# B&R Automation Studio project brse_dtf
Automation Studio 6.5.0.306; technology packages: OpcUaCs 6.5.0

## Configuration ARM

CPU X20CP0484, AutomationRuntime 6.5.1, Build 11.3.0, Vc 6.0.0

### Hardware
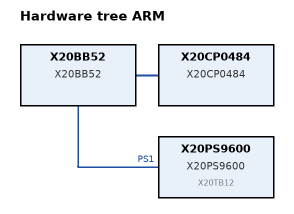
```
X20BB52 : X20BB52 v1.2.0.0
X20CP0484 : X20CP0484 v1.8.1.0  [SL -> X20BB52.SL1]
  TimerDeviceType = SWIOTIMER
  Cyclic1Duration = 10000
  Cyclic1Tolerance = 10000
  Cyclic2Duration = 20000
  Cyclic2Tolerance = 20000
  Cyclic3Duration = 50000
  Cyclic3Tolerance = 50000
  Cyclic4Duration = 100000
  Cyclic4Tolerance = 100000
  Cyclic5Duration = 200000
  Cyclic5Tolerance = 200000
  Cyclic6Duration = 500000
  Cyclic6Tolerance = 500000
  Cyclic7Duration = 1000000
  Cyclic7Tolerance = 1000000
  Cyclic8Duration = 10000
  Cyclic8Tolerance = 30000000
  FileDevice1
  FileDeviceName1 = USER
  FileDevicePath1 = USER_PATH
X20PS9600 : X20PS9600 v1.6.2.0  [PS -> X20BB52.PS1; SS1 -> X20TB12.SS]
X20TB12 : X20TB12 v1.0.0.0
```

## Configuration TS_UnitTest_Sample

CPU , AutomationRuntime 6.5.1, Build 11.3.0

### Task classes (Cpu.sw)
```
Cyclic#4 (cycle 10000 us, tolerance 10000000 us):
  ut_brse_sa <- TS_UnitTest.brse_sandbox_unittest.ut_brse_sandbox.prg
Binaries: udbdef, TCData, iomap, asfw, arconfig, ashwd, sysconf, UaCsConfig, ashwac
Libraries: Runtime, sys_lib, AsIecCon, astime, AsARCfg, AsBrStr, UnitTest, LibAssert1, UtWs, UtMgr, SPLMyCalc, UaCore
```

### Hardware
```
PC_any : PC_any v1.1.2.0 (OrderNumber=PC)
  Cyclic1Duration = 100000
  Cyclic1Tolerance = 10000000
  Cyclic2Duration = 200000
  Cyclic2Tolerance = 10000000
  Cyclic3Duration = 500000
  Cyclic3Tolerance = 10000000
  Cyclic4Duration = 10000
  Cyclic4Tolerance = 10000000
  Cyclic5Duration = 2000000
  Cyclic5Tolerance = 10000000
  Cyclic6Duration = 3000000
  Cyclic6Tolerance = 12000000
  Cyclic7Duration = 4000000
  Cyclic7Tolerance = 12000000
  Cyclic8Duration = 5000000
  Cyclic8Tolerance = 30000000
  ActivateWebServer = 1
```

## Configuration i686

CPU X20CP1686X, AutomationRuntime 6.5.1, Build 11.3.0, Vc 6.5.0

### Task classes (Cpu.sw)
```
Cyclic#4:
  Memleak <- HardwareTest.MemoryLeak.Memleak.prg
  FunctionNa <- HardwareTest.Function.FunctionName.prg
```

### Hardware
```
X20CP1686X : X20CP1686X v1.9.0.0
  FileDevice1
  FileDeviceName1 = USER
  FileDevicePath1 = USER_PATH
```

## Configuration x86_64

CPU PC_any, AutomationRuntime 6.5.1, Build 11.3.0, Vc 6.0.0

### Task classes (Cpu.sw)
```
Cyclic#1:
  FunctionNa <- HardwareTest.Function.FunctionName.prg
  Memleak <- HardwareTest.MemoryLeak.Memleak.prg
Libraries: AsBrStr, AsARCfg, runtime, sys_lib, brse_dtf, astime
```

### Hardware
```
PC : PC_any v1.1.2.0 (OrderNumber=PC)
  FileDevice1
  FileDeviceName1 = USER
  FileDevicePath1 = USER_PATH
```

## Logical view

Binary libraries used (declarations not repeated): operator, runtime, AsIecCon, astime, AsBrStr, AsARCfg, sys_lib, UtMgr 6.5.0, UtWs 6.5.0


### Library Logical/TS_UnitTest/Libraries/UnitTest (ANSIC, version 6.5.0) - Static library for UnitTest programs written in ANSI C /C++

#### UnitTest.h
```c
/*****************************************************************************
 * COPYRIGHT (C) BERNECKER + RAINER
 *****************************************************************************
 * Library:  UnitTest
 * File:     UnitTest.h
 * Author:   B+R
 *****************************************************************************
 * Description: Static library for UnitTest programs written in ANSI C /C++
 *
 * Add the path "\Logical\TS_UnitTest\Libraries\UnitTest\" to the
 * "Additional include directories" in the tab "Build" (PLC Properties)
 ******************************************************************************/

#ifndef	__UNITTEST_H__
#define	__UNITTEST_H__
#ifdef __cplusplus
extern "C"
{
#endif
#include <bur/plctypes.h>

#ifndef NULL
#define	NULL	0
#endif
#include "include/Test.h"

#include "include/TestCase.h"
#include "include/TestListener.h"
#include "include/TestResult.h"
#include "include/TestCaller.h"

#include "include/AssertImpl.h"
#include "include/HelperMacro.h"
#include "include/utRunner.h"

/* function is a test case */
#define _TEST 			static testStatusEnum

/* function is a setup */
#define _SETUP_TEST 	static testStatusEnum 	setupTest

/* function is a teardown */
#define _TEARDOWN_TEST 	static testStatusEnum 	teardownTest

/* function is a setup for whole test set */
#define _SETUP_SET		static testStatusEnum	setupSet

/* function is a teardown for whole test set */
#define _TEARDOWN_SET 	static testStatusEnum	teardownSet

/* function is a cyclic handler for test set */
#define _CYCLIC_SET		static void 			cyclicSetCaller

/* Skipped test case */
#define SKIP_TEST  		_TEST
/* Skip all test cases of set */
#define SKIP_TEST_SET

/* Dummies for smart edit autocompletion.
See AssertImpl.h for real macros used by the compiler  */
#ifdef _SMART_EDIT_DUMMY_

/* String comparison.
Returns true if the strings are equal. */
BOOL TEST_ASSERT_EQUAL_STRING(char *expected,char  *actual);
/* Wstring comparison.
Returns true if the WSTRINGS are equal. */
BOOL TEST_ASSERT_EQUAL_WSTRING(unsigned short *expected,unsigned short *actual);
 /* Compares two memory blocks.
Returns true if [size] bytes are equal. */
BOOL TEST_ASSERT_EQUAL_MEM(void *expected, void *actual,UDINT size);
/* Compares integer values. Usable for all integer types.
Avoid comparison of unsigned with signed types.
Returns true if they are equal.
Note: If different, values are reported as DINT values in the test report */
BOOL TEST_ASSERT_EQUAL_INT(expected, actual);

/* Compares REAL values with delta = (expected * TEST_FLOAT_PRECISION).
Returns true if (difference <= delta) */
BOOL TEST_ASSERT_EQUAL_REAL(REAL expected,REAL actual);
/* Compares REAL values with explicit delta.
Returns true if (difference <= delta) */
BOOL TEST_ASSERT_REAL_WITHIN(REAL delta, REAL expected, REAL actual);
/* Compares LREAL values with delta = (expected * TEST_DOUBLE_PRECISION).
Returns true if (difference <= delta) */
BOOL TEST_ASSERT_EQUAL_LREAL(LREAL expected,LREAL  actual);
/* Compares LREAL values with explicit delta.
Returns true if (difference <= delta) */
BOOL TEST_ASSERT_LREAL_WITHIN(LREAL delta, LREAL expected, LREAL actual);

/* Compares float values with delta = (expected * TEST_FLOAT_PRECISION).
Returns true if (difference <= delta) */
BOOL TEST_ASSERT_EQUAL_FLOAT(float expected, float actual);
/* Compares float values with explicit delta.
Returns true if (difference <= delta) */
BOOL TEST_ASSERT_FLOAT_WITHIN(float delta, float expected, float actual);
/* Compares double values with delta = (expected * TEST_DOUBLE_PRECISION).
Returns true if (difference <= delta) */
BOOL TEST_ASSERT_EQUAL_DOUBLE(double expected, double actual);
/* Compares double values with explicit delta.
Returns true if (difference <= delta) */
BOOL TEST_ASSERT_DOUBLE_WITHIN(double delta, double expected, double actual);

/* Returns true if pointer is null */
BOOL TEST_ASSERT_NULL(void *pointer);
/* Returns true if pointer is not null */
BOOL TEST_ASSERT_NOT_NULL(void *pointer);
/* Returns true, if condition evals to  true */
BOOL TEST_ASSERT_MESSAGE(condition, char *message);
/* Returns true, if condition evals to  true */
BOOL TEST_ASSERT(condition);

/* Returns always false */
BOOL TEST_FAIL(char *message);

/* Add a note to the test report */
void TEST_INFO(char *message);
/* Add a note with location information to the test report */
void TEST_INFO_POS(char *message);

#ifdef __cplusplus
/* Test if expression throws given exception.
Catches all other exceptions as failure.
Note: Available for C++ only */
void TEST_ASSERT_THROW(expression, type);

/* Fails if expression throws any exceptions.
Note: Available for C++ only*/
void TEST_ASSERT_NO_THROW(expression);
#endif

/* Adds a test function with description to the Testfixture.
See UNITTEST_FIXTURES() */
void new_TestFixture(char *name, _TEST function);

/* Adds a test function with description to the Testfixture.
This test will be skipped
See UNITTEST_FIXTURES() */
void skipTestFixture(char *name, _TEST function);

/* Defines the order of test cases.
Should look like this
UNITTEST_FIXTURES(fixtures)
{
	new_TestFixture("test_1",test_1),
	new_TestFixture("test_2",test_2),
	new_TestFixture("test_3",test_3)
}
*/
void UNITTEST_FIXTURES(fixtures)

/* Standard UnitTest caller without any setup / teardown methods*/
void UNITTEST_CALLER_TEST(caller, char *name, fixtures);

/* Standard UnitTest caller with macro setup / teardown for tests*/
void UNITTEST_CALLER_BASIC(caller, char *name, fixtures);

/* UnitTest caller with macro setup / teardown for tests and test set */
void UNITTEST_CALLER_SET(caller, char *name, fixtures);

/* UnitTest caller with macro setup / teardown for tests and test set and cylic*/
void UNITTEST_CALLER_COMPLETE(caller, char *name, fixtures);

/* UnitTest caller with explicit setup / teardown for suite */
void UNITTEST_CALLER_SET_EXPLICIT(caller,name,setupTest,teardownTest,fixtures, setupSuite, teardownSuite);

/* UnitTest caller with explicit setup / teardown for suite and cylic */
void UNITTEST_CALLER_COMPLETE_EXPLICIT(caller,name,setupTest,teardownTest,fixtures, setupSuite, teardownSuite, cyclicCaller);

/* Adds a test set with description to the fixture of test sets.
See UNITTEST_TESTSET_FIXTURES() */
void new_TestSet(testcaller);

/* Defines the order of test sets.
Should look like this
UNITTEST_TESTSET_FIXTURES(fixtures)
{
	new_TestSet(testSet_1),
	new_TestSet(testSet_2),
	new_TestSet(testSet_3)
}*/
void UNITTEST_TESTSET_FIXTURES(fixtures);

/* Defines the test set list handling structure*/
void UNTITTEST_TESTSET_HANDLER();

#endif /*_SMART_EDIT_DUMMY_*/

/*
 Use to declare Test set for use in list of test sets of test programm
 See usage in autogeneratedFile.c / FixtureOfTestSets.c
*/
#define UNITTEST_TESTSET_DECLARATION 	extern const TestCaller

/* Default factor for precision used to test if REAL / float values  are equal.
(0.00001f) */
#define TEST_FLOAT_PRECISION 	(0.00001f)
/* Default factor for precision used to test if LREAL / double values  are equal.
(1e - 12f) */
#define TEST_DOUBLE_PRECISION 	(1e-12f)

#if (__GNUC__ != 11) || (__GNUC_MINOR__ != 3) || (__GNUC_PATCHLEVEL__ != 0)
#error UnitTest is compiled with GCC version 11.3.0. To use UnitTest switch GCC version to 11.3.0 or import a different solution package
#endif

#define UNIT_TEST_LIBRARY_VERSION  			"6.5.0"

#ifdef __cplusplus
};
#endif

#include "include/asserts.hpp"

#endif/*__UNITTEST_H__*/
```

### Package Logical/TS_UnitTest/brse_sandbox_unittest - Easy mode: focus on writing tests

### Program Logical/TS_UnitTest/brse_sandbox_unittest/ut_brse_sandbox (ANSIC) - Empty template for use with helper tool

#### variables.var - Name the suite and add PVs for the program
```iecst
(********************************************************************
 * COPYRIGHT --
 ********************************************************************
 * Program: utTemplate_automated
 * File: variables.var
 * Author: -
 * Created: -
 ********************************************************************
 * Local variables of program utTemplate_automated
 ********************************************************************)
(*Describe the test*)
VAR
	Testsuite : UtMgrTestSuite := (Name:='ut_brse_sandbox',Description:='(Optional field)Template for use with helper tool. Reference or add this program in the package "TS_UnitTest_UpdateTestPrograms"',Type:=utMgrTEST_TYPE_C,MetaInformation:='(Optional field):To be filled');
END_VAR
(*Variables used in the tests*)
```

#### autoGeneratedFile.c - Auto generated code - list of all test sets in the program
```c
/*
B+R UnitTest: This is generated code.
Do not edit! Do not move!
Description: UnitTest Testprogramm infrastructure (List of TestSets).
LastUpdated: 2025-12-15 13:49:51Z
By B+R UnitTest Helper Version: 2.0.0.0
*/
#include "UnitTest.h"

UNITTEST_TESTSET_DECLARATION  Set_brse_arl;

UNITTEST_TESTSET_FIXTURES(utTestSets)
{
	new_TestSet(Set_brse_arl),
};
UNTITTEST_TESTSET_HANDLER();
```

#### Set_brse_arl.c
```c
/********************************************************************
 * COPYRIGHT --
 ********************************************************************
 * Program: -
 * Author:
 * Created:
 ********************************************************************
 * Tests for ...
 ********************************************************************/

#include <bur/plctypes.h>

#ifdef _DEFAULT_INCLUDES
#include <AsDefault.h>
#endif

#include "UnitTest.h"

_CYCLIC_SET()
{

	/* TODO:  add code running cyclically while test set is active here */
	return;
}

_SETUP_SET(void)
{
	/* TODO:  add code running before test set here */
	TEST_DONE;
}

_TEARDOWN_SET(void)
{
	/* TODO:  add code running after test set here */
	TEST_DONE;
}

_SETUP_TEST(void)
{
	/* TODO:  add code running before test case here */
	TEST_DONE;
}

_TEARDOWN_TEST(void)
{
	/* TODO:  add code running after test case here */
	TEST_DONE;
}

_TEST testcase1(void)
{

	/* TODO:  add assertions here */

	/* test is done */
	TEST_ASSERT_EQUAL_INT(3, 1);
	TEST_DONE;
}

_TEST testcase2(void)
{

	/* TODO:  add assertions here */

	/* test is done */
	TEST_ASSERT_EQUAL_INT(3, 3);
	TEST_DONE;
}

/*
B+R UnitTest: This is generated code.
Do not edit! Do not move!
Description: UnitTest Testprogramm infrastructure (TestSet).
LastUpdated: 2025-12-15 13:53:02Z
By B+R UnitTest Helper Version: 2.0.0.0
*/
UNITTEST_FIXTURES(fixtures)
{
	new_TestFixture("testcase1", testcase1),
	new_TestFixture("testcase2", testcase2),
};

UNITTEST_CALLER_COMPLETE_EXPLICIT(Set_brse_arl, "Set_brse_arl", setupTest, teardownTest, fixtures, setupSet, teardownSet, cyclicSetCaller);
```

- find_obsolete_libs.py (not shown)

### obsolete_matches_report.txt
```
No obsolete library matches found.
```

- obsoleteLibs.json (not shown)

### Library Logical/brse_dtf (ANSIC, version 1.11.0) - Library for converting DATE_AND_TIME to and from STRING[50] with a specified format
Depends on: sys_lib, AsBrStr, astime

#### brse_dtf.typ - Exported data types
```iecst
TYPE
	BRSE_DTF_DateTime_typ : 	STRUCT
		start : USINT;
		length : USINT;
	END_STRUCT;
	BRSE_DTF_DateTimeFormat_typ : 	STRUCT  (*Structure describing where to put the values of the date&time at the beginning of the log entry*)
		format : STRING[BRSE_DTF_MAX_LENGTH_STRING];
		year : BRSE_DTF_DateTime_typ;
		month : BRSE_DTF_DateTime_typ;
		day : BRSE_DTF_DateTime_typ;
		hour : BRSE_DTF_DateTime_typ;
		minute : BRSE_DTF_DateTime_typ;
		second : BRSE_DTF_DateTime_typ;
	END_STRUCT;
END_TYPE
```

#### brse_dtf.var - Exported constants
```iecst
VAR CONSTANT
	BRSE_DTF_ERR_FORMAT : UINT := 53902; (*Unexpected date time format*)
	BRSE_DTF_ERR_INPUT : UINT := 53901; (*Input pointer zero*)
	BRSE_DTF_CENTURY_OFFSET : UINT := 2000; (*09 - 02 - 23 --> 2009 - 02 - 23*)
	BRSE_DTF_MAX_LENGTH_STRING : UINT := 50; (*user defined max length of the format/output string*)
END_VAR
```

#### brse_dtf.fun - Exported functions and function blocks
```iecst
FUNCTION BRSE_DTF_CreateFormat : UINT (*Parse a format string and fill the format structure*)
	VAR_INPUT
		pFormatString : UDINT; (*String format*)
		pFormat : UDINT; (*Pointer to a BRSE_DTF_DateTimeFormat_typ*)
	END_VAR
END_FUNCTION

FUNCTION BRSE_DTF_DTToString : UINT (*Returns error code, 0=no error*)
	VAR_INPUT
		DT1 : DATE_AND_TIME; (*32 bit date time in seconds since 1970*)
		pFormat : UDINT; (*Pointer to a BRSE_DTF_DateTimeFormat_typ, created by BRSE_DTF_CreateDateTimeFormat*)
		pStringOutput : UDINT; (*Pointer to formatted string.*)
	END_VAR
END_FUNCTION

FUNCTION BRSE_DTF_StringToDT : UINT (*Returns error code, 0=no error*)
	VAR_INPUT
		pString : UDINT; (*Pointer to formatted string.*)
		pFormat : UDINT; (*Pointer to a BRSE_DTF_DateTimeFormat_typ, created by BRSE_DTF_CreateDateTimeFormat*)
		pDTOutput : UDINT; (*Pointer to return date time value (seconds since 1970)*)
	END_VAR
END_FUNCTION
```

#### brse_dtf_main.h
```c
/*! \file brse_csv_main.h */

/*! \mainpage BRSE_DTF
	\section Introduction

	BRSE_DTF (Date Time Format) is a library used for converting DATE_AND_TIME variables into readable strings via a defined format.

	\arg The format is put together by Y=year (1970-2099), M=month (1-12), D=day (1-31), h=hour (0-23), m=minute (0-59), s=second (0-59).

	\arg A common example is: YYYY-MM-DD hh:mm:ss.

	\arg A format (BRSE_DTF_DateTimeFormat_typ) is created from the format string. This format structure is then used to convert DATE_AND_TIME variables to and from a string value.

	\par Important
	Always use the \b BRSE_DTF_MAX_LENGTH_STRING as length for your format string, as well as for your output strings.
	The library will not take care of limiting the string output to something smaller than this length!

	See an \ref Example on how to use the library.

*/
#include <bur/plctypes.h>
#include <AsBrStr.h>
#include <string.h> /*this will override the asstring functions*/
#include <sys_lib.h>
#include "BRSE_DTF.h"
```

#### brse_dtf.c
```c
/*! \file brse_csv_main.h */

#include "brse_dtf_main.h"

/************************************************************************
  _____                _          __                           _
 / ____|              | |        / _|                         | |
| |     _ __ ___  __ _| |_ ___  | |_ ___  _ __ _ __ ___   __ _| |_
| |    | '__/ _ \/ _` | __/ _ \ |  _/ _ \| '__| '_ ` _ \ / _` | __|
| |____| | |  __/ (_| | ||  __/ | || (_) | |  | | | | | | (_| | |_
 \_____|_|  \___|\__,_|\__\___| |_| \___/|_|  |_| |_| |_|\__,_|\__|
*************************************************************************/

#define START_END_FORMAT(_item_, _strdesc_) 	\
	pSeek = pStrFormat;							\
	length = strcspn(pSeek,_strdesc_);			\
												\
	if(length < strlen(pSeek))					\
	{	pFormat->_item_.start = length;			\
		pSeek+=length;							\
		length = strspn(pSeek,_strdesc_);		\
												\
		pFormat->_item_.length = length;		\
	}											\
	else										\
	{											\
		pFormat->_item_.start = 0;				\
		pFormat->_item_.length = 0;				\
	}

/*! \interface BRSE_DTF_CreateFormat
	\brief Create a date time format from a format string (like YYYY-MM-DD hh:mm:ss).

	This function parametrizes the format structure which is used as an input
	to BRSE_DTF_DTToString and BRSE_DTF_StringToDT. You set a string which defines
	how your output string will look like.
	\par Note
	If you use only two characters for the year in the format YY, the library will assume
	that you mean a year past 2000. You could change this by setting BRSE_DTF_CENTURY_OFFSET to zero.

	\param pFormatString Pointer to the string
	\param pFormat Pointer to BRSE_DTF_DateTimeFormat_typ, the resulting format.
	\retval 0 if successful.
	\retval BRSE_DTF_ERR_INPUT if one of the input pointers are zero
*/
UINT BRSE_DTF_CreateFormat(UDINT formatStringAddress, UDINT formatAddress)
{
	BRSE_DTF_DateTimeFormat_typ *pFormat;
	char 	*pStrFormat;
	char	*pSeek;
	UINT 	length;

	if (formatStringAddress == 0 || formatAddress == 0)
		return BRSE_DTF_ERR_INPUT;

	pFormat = (BRSE_DTF_DateTimeFormat_typ *)formatAddress;
	pStrFormat = (char *)formatStringAddress;

	strncpy(pFormat->format,pStrFormat,BRSE_DTF_MAX_LENGTH_STRING);

	START_END_FORMAT( year, 	"Y" );
	START_END_FORMAT( month, 	"M" );
	START_END_FORMAT( day, 		"D" );
	START_END_FORMAT( hour, 	"h" );
	START_END_FORMAT( minute, 	"m" );
	START_END_FORMAT( second, 	"s" );

	return 0;
}

/*************************************************************************
 _______       _____ _        _
|__   __|     / ____| |      (_)
   | | ___   | (___ | |_ _ __ _ _ __   __ _
   | |/ _ \   \___ \| __| '__| | '_ \ / _` |
   | | (_) |  ____) | |_| |  | | | | | (_| |
   |_|\___/  |_____/ \__|_|  |_|_| |_|\__, |
                                       __/ |
                                      |___/
*************************************************************************/
#define COPY_DATE_TIME(_item_) 					\
	brsitoa(pTime->_item_,(UDINT)ascii_val);		\
	length = strlen(ascii_val);					\
	offset = 0;									\
	startoffset = 0;							\
												\
	if(length > pFormat->_item_.length)			\
	{											\
		/*eg. YY is specified and year is 1981 */\
		offset = length - pFormat->_item_.length;\
		/*start with ascii_val[offset]*/ 		\
		length = pFormat->_item_.length;		\
	}											\
	else if(length < pFormat->_item_.length)	\
	{											\
		/*lets say month is 9, and MM is specified*/\
		startoffset = pFormat->_item_.length - length;\
		/*start copying one character later*/	\
	}											\
												\
	memset(pStr + pFormat->_item_.start,'0',pFormat->_item_.length);/*insert leading zeros to make it 2005-05-05 instead of 2005- 5 - 5*/\
	memcpy(pStr + pFormat->_item_.start + startoffset ,&ascii_val[offset],length);

/*! \interface BRSE_DTF_DTToString
	\brief Convert a DATE_AND_TIME value to string using a certain created format.

	\param DT1 DATE_AND_TIME to convert.
	\param pFormat Pointer to BRSE_DTF_DateTimeFormat_typ, the format to use.
	\param pStringOutput Pointer to the resulting string.
	\retval 0 if successful.
	\retval BRSE_DTF_ERR_INPUT if one of the input pointers are zero
*/
UINT BRSE_DTF_DTToString(DATE_AND_TIME dt, UDINT formatAddress, UDINT stringOutputAddress)
{
	char *pStr = 0;
	BRSE_DTF_DateTimeFormat_typ *pFormat = 0;
	DTStructure dtStruct;
	DTStructure *pTime = &dtStruct;
	char ascii_val[15];
	UDINT length,offset,startoffset;

	if (formatAddress == 0 || stringOutputAddress == 0)
		return BRSE_DTF_ERR_INPUT;

	memset(&dtStruct, 0, sizeof(dtStruct));
	DT_TO_DTStructure(dt, (UDINT)&dtStruct);
	pStr = (char *)stringOutputAddress;
	pFormat = (BRSE_DTF_DateTimeFormat_typ *)formatAddress;

	strncpy(pStr,pFormat->format,BRSE_DTF_MAX_LENGTH_STRING);

	COPY_DATE_TIME(year);
	COPY_DATE_TIME(month);
	COPY_DATE_TIME(day);
	COPY_DATE_TIME(hour);
	COPY_DATE_TIME(minute);
	COPY_DATE_TIME(second);

	return 0;
}

/**************************************************************************
 ______                      _____ _        _
|  ____|                    / ____| |      (_)
| |__ _ __ ___  _ __ ___   | (___ | |_ _ __ _ _ __   __ _
|  __| '__/ _ \| '_ ` _ \   \___ \| __| '__| | '_ \ / _` |
| |  | | | (_) | | | | | |  ____) | |_| |  | | | | | (_| |
|_|  |_|  \___/|_| |_| |_| |_____/ \__|_|  |_|_| |_|\__, |
                                                     __/ |
                                                    |___/
*************************************************************************/

#define PARSE_DATE_TIME(_item_) 				\
												\
	memset(&ascii_val[0], 0, sizeof(ascii_val));\
	memcpy(&ascii_val[0], pStr + pFormat->_item_.start, pFormat->_item_.length);\
	for (i=0; i<pFormat->_item_.length; i++)	\
	{											\
		if (ascii_val[i] < 0x30 || ascii_val[i] > 0x39)\
		{										\
			return BRSE_DTF_ERR_FORMAT;			\
		}										\
	}											\
	pTime->_item_ = brsatoi((UDINT)&ascii_val[0]);

/*! \interface BRSE_DTF_StringToDT
	\brief Parse a string to DATE_AND_TIME value using a certain created format.

	\param pString string to parse.
	\param pFormat Pointer to BRSE_DTF_DateTimeFormat_typ, the format to use.
	\param pDTOutput Pointer to the resulting DATE_AND_TIME object.
	\retval 0 if successful.
	\retval BRSE_DTF_ERR_INPUT if one one the input pointers are zero
	\retval BRSE_DTF_ERR_FORMAT if the input string does not give a valid date
*/
UINT BRSE_DTF_StringToDT(UDINT stringAddress, UDINT formatAddress, UDINT dateTimeOutputAddress)
{
	char *pStr = 0;
	DTStructure dtStruct;
	DTStructure *pTime = &dtStruct;
	BRSE_DTF_DateTimeFormat_typ *pFormat= 0;
	DATE_AND_TIME dt = 0;
	char ascii_val[15];
	int i = 0;
	if (stringAddress == 0 || formatAddress == 0)
		return BRSE_DTF_ERR_INPUT;

	pStr = (char *)stringAddress;
	pFormat = (BRSE_DTF_DateTimeFormat_typ *)formatAddress;

	memset(&dtStruct, 0, sizeof(dtStruct));
	PARSE_DATE_TIME(year);
	PARSE_DATE_TIME(month);
	PARSE_DATE_TIME(day);
	PARSE_DATE_TIME(hour);
	PARSE_DATE_TIME(minute);
	PARSE_DATE_TIME(second);

	if (pFormat->year.length > 0 && dtStruct.year < 1970) /* add current year */
		dtStruct.year += BRSE_DTF_CENTURY_OFFSET;

	/* set default valuess where 0 is not accepted */
	if (dtStruct.year == 0)
		dtStruct.year = 1970;
	if (dtStruct.month == 0)
		dtStruct.month = 1;
	if (dtStruct.day == 0)
		dtStruct.day = 1;

	dt = DTStructure_TO_DT((UDINT)&dtStruct);

	if((UDINT)dt == 0xFFFFFFFF) return BRSE_DTF_ERR_FORMAT;

	memcpy((DATE_AND_TIME *)dateTimeOutputAddress, &dt, sizeof(dt));
	return 0;
}
```

#### version_history.c
```c
/*!

\page History

\section History

\par V1.00
\arg First version.

\par V1.10
\arg BRSE_DTF_StringToDT Added status ouput BRSE_DTF_ERR_INPUT when the date and time was outside valid bounds, eg. september 31st
\arg BRSE_DTF_CreateFormat now also saving the format string into the structure
\arg BRSE_DTF_DTToString Changed so that the format string is copied to the output string before copying the values

\par V1.11
\arg Library dependency has been changed from AsString to AsBrStr, so that conflicts can be avoided with ANSI-C standard functions(atof, atoi etc.)
*/
```

#### example.c
```c
/*!

\page Example
\anchor Example

\section Example
This example shows how to convert between DATE_AND_TIME and STRING variables using the DTF library.

<a href = "y:\Application\Libraries\BRSE_DTF\Documentation\ConvertDate.zip" >Get the ZIP Import Package for AS3</a>

\par ConvertDate.typ
\code
TYPE
	ConvertDate_typ : 	STRUCT
		Address : UDINT;
		Input : ConvertDateInput_typ;
		Output : ConvertDateOutput_typ;
	END_STRUCT;
	ConvertDateInput_typ : 	STRUCT
		Command : ConvertDateInputCommand_typ;
		Format : STRING[BRSE_DTF_MAX_LENGTH_STRING];
		DataAsString : STRING[BRSE_DTF_MAX_LENGTH_STRING];
		DataAsDateTime : DATE_AND_TIME;
	END_STRUCT;
	ConvertDateInputCommand_typ : 	STRUCT
		ConvertToString : USINT;
		ConvertToDateTime : USINT;
	END_STRUCT;
	ConvertDateOutput_typ : 	STRUCT
		ConvertedToDateTime : DATE_AND_TIME;
		ConvertedToString : STRING[BRSE_DTF_MAX_LENGTH_STRING];
		Status : UINT;
	END_STRUCT;
END_TYPE
\endcode

\par ConvertDate.var
\code
VAR
	ConvertDate : ConvertDate_typ;
	ConversionFormat : BRSE_DTF_DateTimeFormat_typ;
END_VAR
\endcode

\par ConvertDate.st
\code
PROGRAM _INIT

	ConvertDate.Address := ADR(ConvertDate);

	ConvertDate.Input.Format := 'YYYY-MM-DD hh:mm:ss';

END_PROGRAM

PROGRAM _CYCLIC

	(*convert STRING[50] to DATE_AND_TIME*)
	IF ConvertDate.Input.Command.ConvertToDateTime <> 0 THEN

		ConvertDate.Output.Status := BRSE_DTF_CreateFormat(
			ADR(ConvertDate.Input.Format),
			ADR(ConversionFormat));

		IF ConvertDate.Output.Status <> 0 THEN RETURN; END_IF

		ConvertDate.Output.Status := BRSE_DTF_StringToDT(
			ADR(ConvertDate.Input.DataAsString),
			ADR(ConversionFormat),
			ADR(ConvertDate.Output.ConvertedToDateTime));

		ConvertDate.Input.Command.ConvertToDateTime := 0;

	END_IF

	(*convert DATE_AND_TIME to STRING[50]*)
	IF ConvertDate.Input.Command.ConvertToString <> 0 THEN

		ConvertDate.Output.Status := BRSE_DTF_CreateFormat(
			ADR(ConvertDate.Input.Format),
			ADR(ConversionFormat));

		IF ConvertDate.Output.Status <> 0 THEN RETURN; END_IF

		ConvertDate.Output.Status := BRSE_DTF_DTToString(
			ConvertDate.Input.DataAsDateTime,
			ADR(ConversionFormat),
			ADR(ConvertDate.Output.ConvertedToString));

		ConvertDate.Input.Command.ConvertToString := 0;

	END_IF

END_PROGRAM
\endcode

*/
```

Listed in the project but not available here: Logical/Global.typ, Logical/Global.var, Logical/TS_UnitTest/Libraries/UnitTest/include, Logical/TS_UnitTest/Libraries/UnitTest/src, Logical/TS_UnitTest/Samples, Logical/TS_UnitTest/Templates/HelperTool_Supported, Logical/TS_UnitTest/Templates/NoToolSupport, Logical/TS_UnitTest/brse_sandbox_unittest/ut_brse_sandbox/testSuite.c, Logical/TS_UnitTest/brse_sandbox_unittest/TestSet_Templates, Logical/HardwareTest/MemoryLeak/Memleak, Logical/HardwareTest/Function/FunctionName
